PROGRAM PRG_TEST
VAR
	fbSum_Test : FB_Sum_Test;
END_VAR

TcUnit.RUN();

END_PROGRAM

(* stored: Version 1.1.0.1, ProductVersion 3.1.4022.18
   POU PRG_TEST: Id {e571d8c7-b2e6-40a1-b02a-f04440559a76}, SpecialFunc None *)
